{attribute 'linkalways'} 
{attribute 'no_explicit_call' := 'This FB is a CLASS and must be accessed using methods or properties'}
{attribute 'enable_dynamic_creation'}
FUNCTION_BLOCK _LWORD EXTENDS NumericDatatypeBase
VAR
	localData : LWORD;
	activeData : REFERENCE TO LWORD REF= localData;
END_VAR

PROPERTY PUBLIC Address : PVOID
GET
Address := ADR(activeData);
END_GET
END_PROPERTY

METHOD PUBLIC ClearReference
VAR_INPUT
END_VAR
activeData REF= localData;
END_METHOD

METHOD PUBLIC Clone : I_Datatype
VAR
    pClone : POINTER TO _LWORD;
END_VAR
pClone := __NEW(_LWORD(InitialValue := Value));
Clone := pClone^;
END_METHOD

METHOD FB_init : BOOL
VAR_INPUT
	bInitRetains : BOOL; // if TRUE, the retain variables are initialized (warm start / cold start)
	bInCopyCode : BOOL;  // if TRUE, the instance afterwards gets moved WORDo the copy code (online change)
	InitialValue : LWORD;
END_VAR
localData := InitialValue;
END_METHOD

PROPERTY PUBLIC IsFloat : BOOL
GET
IsFloat := FALSE;
END_GET
END_PROPERTY

PROPERTY PUBLIC IsSigned : BOOL
GET
IsSigned := FALSE;
END_GET
END_PROPERTY

PROPERTY PUBLIC LowerBound : LWORD
GET
LowerBound := DatatypeLimits.LWORD_LOWER_LIMIT;
END_GET
END_PROPERTY

METHOD PUBLIC MakeReferenceTo
VAR_INPUT
	ReferenceTarget : REFERENCE TO LWORD;
END_VAR
activeData REF= ReferenceTarget;
END_METHOD

METHOD PROTECTED SerializeLowerbound
VAR_INPUT
	Serializer : I_Serializer;
END_VAR
Serializer.AddLword(Lowerbound);
END_METHOD

METHOD PROTECTED SerializeUpperbound
VAR_INPUT
	Serializer : I_Serializer;
END_VAR
Serializer.AddLword(Upperbound);
END_METHOD

METHOD PUBLIC SerializeWith
VAR_INPUT
	Serializer : I_Serializer;
END_VAR
Serializer.AddLword(activeData);
END_METHOD

PROPERTY PUBLIC Size : UDINT
GET
Size := SIZEOF(activeData);
END_GET
END_PROPERTY

METHOD TryDeserializeFrom : BOOL
VAR_INPUT
	Deserializer : I_Deserializer;
	Feedback : I_DeserializerFeedback;
END_VAR
TryDeserializeFrom := Deserializer.TryGetLword(activeData, Feedback);
END_METHOD

METHOD TryMakeReferenceTo : BOOL
VAR_INPUT
	Target : I_Datatype;
END_VAR
VAR
	pTargetData : POINTER TO LWORD;
END_VAR
IF NOT (Target.TypeName = TypeName) THEN
	RETURN;
END_IF

pTargetData := Target.Address;
activeData REF= pTargetData^;
TryMakeReferenceTo := TRUE;
END_METHOD

PROPERTY PUBLIC TypeName : T_MAXSTRING
GET
TypeName := 'LWORD';
END_GET
END_PROPERTY

PROPERTY PUBLIC UpperBound : LWORD
GET
UpperBound :=  DatatypeLimits.LWORD_UPPER_LIMIT;
END_GET
END_PROPERTY

PROPERTY PUBLIC Value : LWORD
GET
Value := activeData;
END_GET
SET
activeData := Value;
END_SET
END_PROPERTY

END_FUNCTION_BLOCK

(* stored: Version 1.1.0.1, ProductVersion 3.1.4024.12
   POU _LWORD: Id {602f8844-fe02-0e80-0b36-323dce08983e}, SpecialFunc None
   Folder Constructor: Id {5117c729-ea46-064c-2b01-911326316470}
   Folder Protected: Id {1be7b19c-2e2e-0bd3-3b01-8cbc4b73dcdc}
   Property Address: Id {c3e72b9b-b305-0ceb-22a7-6f4f6729f1cf}
   Get Get: Id {525ba87c-0806-02d3-1e4f-be7970cef05e}
   Method ClearReference: Id {34206305-7c53-08d0-0d5d-4437b9f74319}
   Method Clone: Id {9988e23c-5d3c-02f6-3725-a895be3ad589}
   Method FB_init: Id {48f7bf04-c509-0a15-240d-51246c245ad9}
   Property IsFloat: Id {2e224b9d-7970-0bce-2bae-444bfab1cc8b}
   Get Get: Id {92861380-9f26-0950-0d71-a25da5a378ef}
   Property IsSigned: Id {6f27144c-e414-0e68-3f1b-cc10e428a86a}
   Get Get: Id {bc0165a3-18b5-0557-1588-350d720409e9}
   Property LowerBound: Id {8e93eb50-1df4-0ef3-1fc1-d0d55d661019}
   Get Get: Id {fc2ae3ce-480f-0d59-393b-3102666a03af}
   Method MakeReferenceTo: Id {12bba3b5-9991-04b9-34a6-933b6ca71bb5}
   Method SerializeLowerbound: Id {91badad0-5a6a-007a-1d16-668f3de518bc}
   Method SerializeUpperbound: Id {eea66163-b09d-0986-1a7a-0ca356dc29b7}
   Method SerializeWith: Id {a268215b-a841-03a3-2176-4db11cf8cc04}
   Property Size: Id {a11fa9fc-83a7-0fec-324a-180acf8de2f0}
   Get Get: Id {339d599c-84ee-0bda-0fa9-40be9479f22b}
   Method TryDeserializeFrom: Id {f55755a7-10ba-0cd9-010f-34002485ad75}
   Method TryMakeReferenceTo: Id {ca0a5ce3-d3dc-0afc-1dd9-09326a75bd45}
   Property TypeName: Id {495ebda8-c10c-0a18-072c-c4ac5e8c3fd3}
   Get Get: Id {507feb5f-b9ae-0c41-3b42-52c461b263b0}
   Property UpperBound: Id {46dc14a8-2164-0dd7-1ba3-df4aca5ac47f}
   Get Get: Id {1b379011-09f2-063d-1fd2-2f947edf507e}
   Property Value: Id {fdfc032e-f89e-07af-037f-a8207d8e0827}
   Get Get: Id {eb611be1-1233-0803-18e2-19c01df2555d}
   Set Set: Id {766d6c12-22d3-0d2b-1f8f-ee17200dbd09} *)
